Universal Robots PolyScope program: all instructions.urp

Program all instructions (installation=default createdIn=5.6.0.90886 lastSavedIn=5.6.0.90886 robotSerialNumber=20195699999)
Robot Program (runOnlyOnce=false)
  Set DigitalOutput pin=digital_out[2]; digitalValue=1
  Wait DigitalInput pin=digital_in[1]; digitalValue=1
  Wait DigitalInput pin=digital_in[4]; digitalValue=0
  Wait Sleep waitTime=1
  MoveL speed 250 mm/s, acceleration 1200 mm/s^2 (useActiveTCP=true) feature=Base
    Waypoint Waypoint_2: motionParameters(jointSpeed=1.047198 jointAcceleration=1.396263 cartesianSpeed=0.25 cartesianAcceleration=1.2); TCP in base x=-184.548 y=-439.731 z=278.361 mm, rx=-0.0012 ry=3.1163 rz=0.0389 rad; joints [-91.713, -98.956, -126.223, -46.295, 91.392, -1.776] deg; TCP offset x=0 y=0 z=0 mm, rx=0 ry=0 rz=0 rad
    Waypoint Waypoint_3: TCP in base x=-184.548 y=-439.731 z=278.361 mm, rx=-0.0012 ry=3.1163 rz=0.0389 rad; joints [-91.713, -98.956, -126.223, -46.295, 91.392, -1.776] deg
    Waypoint Waypoint_4: TCP in base x=-187.384 y=-440.532 z=278.361 mm, rx=-0.0012 ry=3.1163 rz=0.0389 rad; joints [-92.072, -99.161, -125.952, -46.369, 91.383, -2.134] deg; TCP offset x=0 y=0 z=0 mm, rx=0 ry=0 rz=0 rad
  MoveL speed 250 mm/s, acceleration 1200 mm/s^2 (useActiveTCP=true) feature=Base
    Waypoint Waypoint_5 (Relative): relativeFromPosition joints [-91.713, -98.956, -126.223, -46.295, 91.392, -1.776] deg; TCP in base x=-184.548 y=-439.731 z=278.361 mm, rx=-0.005 ry=3.1056 rz=-0.2632 rad; joints [-91.804, -99.669, -131.176, -29.516, 91.739, -1.842] deg
  MoveJ speed 60 deg/s, acceleration 80 deg/s^2 (useActiveTCP=true) feature=Base
    Waypoint Waypoint_1: motionParameters(jointSpeed=1.047198 jointAcceleration=1.396263 cartesianSpeed=0.25 cartesianAcceleration=1.2); TCP in base x=-184.548 y=-439.731 z=278.361 mm, rx=-0.0012 ry=3.1163 rz=0.0389 rad; joints [-91.713, -98.956, -126.223, -46.295, 91.392, -1.776] deg
